(* CODESYS project Prueba_1_RECOVERED_2026-04-10T18-21-56.project

Project tree, tasks and I/O mapping:
  Device : CODESYS Control Win V3 x64, CODESYS, version 3.5.20.20
    application Application
      libraries: Standard, 3.5.18.0 (System)
      task MainTask (cyclic, interval t#20ms, priority 1) calls PLC_PRG
      global variables GVL_IO
      program PLC_PRG [SFC]: IZAJE_ANT_entry, DES_TLK_entry, ACT_TLK_during, CARRO_ANT_entry, DES_TLK_during, TALK_entry, LISTEN_entry, ACT_TLK_entry
  program POU [SFC]
*)

// Device/Application/GVL_IO
{attribute 'qualified_only'}
VAR_GLOBAL
	//Entradas Digitales
	bFC_SUP       AT %IX0.0  : BOOL; // In0
    bFC_INF       AT %IX0.1  : BOOL; // In1
    bFC_IZQ       AT %IX0.2  : BOOL; // In2
    bFC_DER       AT %IX0.3  : BOOL; // In3
	bFalla_E      AT %IX0.4 : BOOL; // In4
	bBalanceo_on  AT %IX0.5 : BOOL; // In5
    bTLK_act      AT %IX0.6 : BOOL; // In6

	//Entradas Analógicas
    rFhw          AT %IW0  : REAL; // In1
    rMI           AT %IW1  : REAL; // In2
    rXtd          AT %IW2  : REAL; // In3
    rWhm          AT %IW3  : REAL; // In4
    rWhm_ant      AT %IW4  : REAL; // In5
    rWtm          AT %IW5  : REAL; // In6
    rWtm_ant      AT %IW6 : REAL; // In7
    rLh           AT %IW7 : REAL; // In8
    rDLh_max      AT %IW8 : REAL; // In9
    rDLh_ref_man  AT %IW9 : REAL; // In10
    rDXt_ref_man  AT %IW10 : REAL; // In11
    rDestino      AT %IW11 : REAL; // In12
    rYc0_xt       AT %IW12 : REAL; // In13
    rY_c0         AT %IW13 : REAL; // In14
    rT_sim        AT %IW14 : REAL; // In15
    rTtm_disp     AT %IW15 : REAL; // In16
    rThm_disp     AT %IW16 : REAL; // In17
	
	//Salidas Digitales
	bTLK 		  AT %QX0.0 : BOOL; // Out1
	bBal_control  AT %QX0.1 : BOOL; // Out2
	bBRK_h		  AT %QX0.2 : BOOL; // Out3
	bBRK_hE		  AT %QX0.3 : BOOL; // Out4
	bBRK_t		  AT %QX0.4 : BOOL; // Out5
	bAlive		  AT %QX0.5 : BOOL; // Out6
	
	//Salidas Analógicas
    rDxt_ref      AT %QW0  : REAL; // Out7
	rDlh_ref      AT %QW1  : REAL; // Out8
	iC		      AT %QW2  : DINT; // Out8
	iMl_estimada  AT %QW1  : DINT; // Out8

END_VAR

// Device/Application/PLC_PRG
PROGRAM PLC_PRG

VAR
	alive: BOOL := 0;
	dxt_ref: REAL := 0;
	dlh_ref: REAL := 0;
	dlh_ref_ant: REAL := 0;
	dxt_ref_ant: REAL := 0;
	op_mode: BOOL := 0;
	cable_tenso: BOOL := 0;
	xtd: REAL := 0;
	y_real: REAL;
	lh: REAL;
	Hc: REAL := 2.54;
	whm: REAL;
	whm_ant: REAL;
	whm_min: LREAL;
	falla_E: BOOL;
	TLK: BOOL := 0;
	c: DINT := 0;
END_VAR
VAR CONSTANT
	Wc: REAL := 2.44;
END_VAR

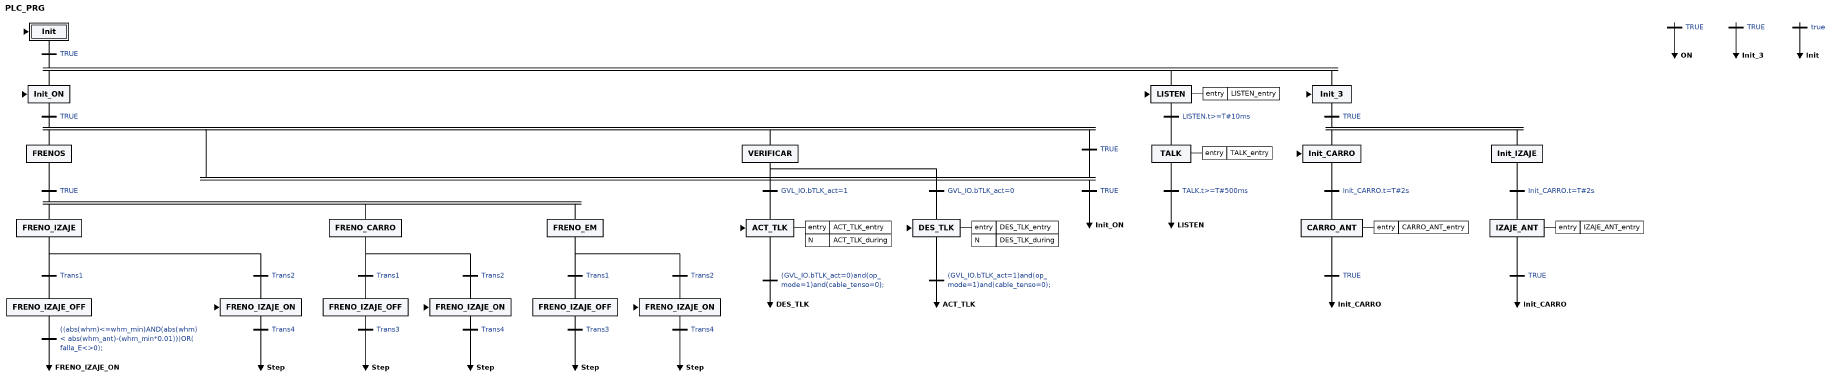
INITIAL_STEP Init:
END_STEP
TRANSITION FROM Init TO (Init_ON, LISTEN, Init_3)
    := TRUE;
END_TRANSITION
// macro ON begins
// macro OFF begins
STEP Init_ON:
END_STEP
TRANSITION FROM Init_ON TO (FRENOS, VERIFICAR, ???, ???, ???)
    := TRUE;
END_TRANSITION
// macro DETECCION_ESTADOS begins
STEP FRENOS:
END_STEP
TRANSITION FROM FRENOS TO (FRENO_IZAJE, FRENO_CARRO, FRENO_EM)
    := TRUE;
END_TRANSITION
STEP FRENO_IZAJE:
END_STEP
TRANSITION FROM FRENO_IZAJE TO FRENO_IZAJE_OFF
    := Trans1;
END_TRANSITION
STEP FRENO_IZAJE_OFF:
END_STEP
TRANSITION FROM FRENO_IZAJE_OFF TO FRENO_IZAJE_ON
    := ((abs(whm)<=whm_min)AND(abs(whm) < abs(whm_ant)-(whm_min*0.01)))OR(falla_E<>0);
END_TRANSITION
TRANSITION FROM FRENO_IZAJE TO FRENO_IZAJE_ON
    := Trans2;
END_TRANSITION
STEP FRENO_IZAJE_ON:
END_STEP
TRANSITION FROM FRENO_IZAJE_ON TO Step
    := Trans4;
END_TRANSITION
STEP FRENO_CARRO:
END_STEP
TRANSITION FROM FRENO_CARRO TO FRENO_IZAJE_OFF
    := Trans1;
END_TRANSITION
STEP FRENO_IZAJE_OFF:
END_STEP
TRANSITION FROM FRENO_IZAJE_OFF TO Step
    := Trans3;
END_TRANSITION
TRANSITION FROM FRENO_CARRO TO FRENO_IZAJE_ON
    := Trans2;
END_TRANSITION
STEP FRENO_IZAJE_ON:
END_STEP
TRANSITION FROM FRENO_IZAJE_ON TO Step
    := Trans4;
END_TRANSITION
STEP FRENO_EM:
END_STEP
TRANSITION FROM FRENO_EM TO FRENO_IZAJE_OFF
    := Trans1;
END_TRANSITION
STEP FRENO_IZAJE_OFF:
END_STEP
TRANSITION FROM FRENO_IZAJE_OFF TO Step
    := Trans3;
END_TRANSITION
TRANSITION FROM FRENO_EM TO FRENO_IZAJE_ON
    := Trans2;
END_TRANSITION
STEP FRENO_IZAJE_ON:
END_STEP
TRANSITION FROM FRENO_IZAJE_ON TO Step
    := Trans4;
END_TRANSITION
STEP VERIFICAR:
END_STEP
TRANSITION FROM VERIFICAR TO ACT_TLK
    := GVL_IO.bTLK_act=1;
END_TRANSITION
STEP ACT_TLK:
    ACT_TLK_entry(P1);  // entry action
    ACT_TLK_during(N);
END_STEP
TRANSITION FROM ACT_TLK TO DES_TLK
    := (GVL_IO.bTLK_act=0)and(op_mode=1)and(cable_tenso=0);
END_TRANSITION
TRANSITION FROM VERIFICAR TO DES_TLK
    := GVL_IO.bTLK_act=0;
END_TRANSITION
STEP DES_TLK:
    DES_TLK_entry(P1);  // entry action
    DES_TLK_during(N);
END_STEP
TRANSITION FROM DES_TLK TO ACT_TLK
    := (GVL_IO.bTLK_act=1)and(op_mode=1)and(cable_tenso=0);
END_TRANSITION
TRANSITION FROM ??? TO ???
    := TRUE;
END_TRANSITION
TRANSITION FROM (???, ???, ???) TO Init_ON
    := TRUE;
END_TRANSITION
TRANSITION FROM ??? TO Init_ON
    := TRUE;
END_TRANSITION
// macro VIVO begins
STEP LISTEN:
    LISTEN_entry(P1);  // entry action
END_STEP
TRANSITION FROM LISTEN TO TALK
    := LISTEN.t>=T#10ms;
END_TRANSITION
STEP TALK:
    TALK_entry(P1);  // entry action
END_STEP
TRANSITION FROM TALK TO LISTEN
    := TALK.t>=T#500ms;
END_TRANSITION
// macro DELAY_VARIABLES begins
STEP Init_3:
END_STEP
TRANSITION FROM Init_3 TO (Init_CARRO, Init_IZAJE)
    := TRUE;
END_TRANSITION
// macro CARRO begins
STEP Init_CARRO:
END_STEP
TRANSITION FROM Init_CARRO TO CARRO_ANT
    := Init_CARRO.t=T#2s;
END_TRANSITION
STEP CARRO_ANT:
    CARRO_ANT_entry(P1);  // entry action
END_STEP
TRANSITION FROM CARRO_ANT TO Init_CARRO
    := TRUE;
END_TRANSITION
// macro IZAJE begins
STEP Init_IZAJE:
END_STEP
TRANSITION FROM Init_IZAJE TO IZAJE_ANT
    := Init_CARRO.t=T#2s;
END_TRANSITION
STEP IZAJE_ANT:
    IZAJE_ANT_entry(P1);  // entry action
END_STEP
TRANSITION FROM IZAJE_ANT TO Init_CARRO
    := TRUE;
END_TRANSITION
TRANSITION FROM ??? TO Init_3
    := TRUE;
END_TRANSITION
TRANSITION FROM ??? TO Init
    := true;
END_TRANSITION

ACTION IZAJE_ANT_entry:
dlh_ref_ant:=dlh_ref;
END_ACTION

ACTION DES_TLK_entry:
TLK:=0;
c:=Trunc((xtd+30/Wc));
END_ACTION

ACTION ACT_TLK_during:
y_real:=45-(lh+Hc);
END_ACTION

ACTION CARRO_ANT_entry:
dxt_ref_ant:=dxt_ref;
END_ACTION

ACTION DES_TLK_during:
y_real:=45-lh;
END_ACTION

ACTION TALK_entry:
alive:=1;
END_ACTION

ACTION LISTEN_entry:
alive:=0;
END_ACTION

ACTION ACT_TLK_entry:
TLK:=1;
c:=-TRUNC((xtd+30)/Wc);
END_ACTION

END_PROGRAM

// POU
PROGRAM POU
VAR
END_VAR

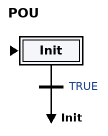
INITIAL_STEP Init:
END_STEP
TRANSITION FROM Init TO Init
    := TRUE;
END_TRANSITION

END_PROGRAM
